Fanuc KAREL source: kf00045.KL

-- PROVISIONAL review KL for V770-1; original PC SHA256 85cda64ff5c6f4a92c3e7fa77a35b2dfee1ee2d25c8ba95c0b96d5874d943797
-- Incomplete behavior may be omitted. Consult companion uncertainty JSON. Do not deploy.
PROGRAM KF00045
%NOLOCKGROUP
VAR
  I : INTEGER
  J : INTEGER
  X : REAL
  Y : REAL
  B : BOOLEAN
  C : BOOLEAN
  TXT : STRING[80]
  TXT2 : STRING[80]
  STATUS : INTEGER
-- UNRESOLVED_DECL AI type=002010
-- UNRESOLVED_DECL BI type=002010
-- UNRESOLVED_DECL P type=000102
-- UNRESOLVED_DECL JP type=000199
-- UNRESOLVED_DECL PF type=000101
-- UNRESOLVED_DECL V1 type=000013
-- UNRESOLVED_DECL V2 type=000013
BEGIN
  -- UNRESOLVED_PC offsets 5-12; opcodes 9D,23
  -- UNRESOLVED_PC offsets 17-30; opcodes 21,9D,57,79
  -- UNRESOLVED_PC offsets 35-49; opcodes 21,9D,52,23
  -- UNRESOLVED_PC offsets 59-63; opcodes 7F
END KF00045
